(* IEC 61131-3 sources: SFWE411-511/ladder-diagrams/PLC/build/build, 2 files *)

(* ---- plc.st ---- *)
TYPE
  LOGLEVEL : (CRITICAL, WARNING, INFO, DEBUG) := INFO;
END_TYPE

FUNCTION_BLOCK LOGGER
  VAR_INPUT
    TRIG : BOOL;
    MSG : STRING;
    LEVEL : LOGLEVEL := INFO;
  END_VAR
  VAR
    TRIG0 : BOOL;
  END_VAR

  IF TRIG AND NOT TRIG0 THEN
  {{
   LogMessage(GetFbVar(LEVEL),(char*)GetFbVar(MSG, .body),GetFbVar(MSG, .len));
  }}
  END_IF;
  TRIG0:=TRIG;
END_FUNCTION_BLOCK

PROGRAM program0
  VAR
    EntranceGateSensor : BOOL;
    EntranceGateSensor0 : BOOL;
    ticketValidationEnter : BOOL;
    ticketValidationExit : BOOL;
    PhysicalCardEnter : BOOL;
    PhysicalCardExit : BOOL;
    PermitCardEnter : BOOL;
    PermitCardExit : BOOL;
    openSpotSensor : BOOL;
    countSensor : BOOL;
    overstayNotification : BOOL;
    OpenEntryGate : BOOL;
    OverstaySignage : BOOL;
    AvailableSpotSignage : BOOL;
    LicensePlateCapture : BOOL;
    LicensePlateVerification : BOOL;
    EntrancePassThrough : BOOL;
    AlarmButton : BOOL;
    TempSensor : BOOL;
    parkingLED : BOOL;
    AlarmActivate : BOOL;
    HealthDisplay : BOOL;
    CloseEntryGate : BOOL;
    LightSensor : INT := 100;
    SetLight : BOOL;
    RainSensor : BOOL;
    SnowSensor : BOOL;
    ClearWeather : BOOL;
    LightControl : BOOL;
    RainSignage : BOOL;
    SnowSignage : BOOL;
    ClearSignage : BOOL;
  END_VAR
  VAR
    ParkingTimer : INT;
    ParkingLimit : INT := 60;
  END_VAR
  VAR
    ParkingDurationStatus : BOOL;
    OverstayDetector : BOOL;
    TicketValidationSensor : BOOL;
    PaymentMachineDisplay : BOOL;
    EVSensorStatus : BOOL;
    EVChargerActivation : BOOL;
    ExitSensor : BOOL;
    ExitPassThroughSensor : BOOL;
    LicensePlateCaptureSystem : WORD;
    ExitGateOpens : BOOL;
    ExitGateCloses : BOOL;
  END_VAR
  VAR
    LightSensorCondition : INT := 10;
  END_VAR
  VAR
    HMIEntryDisplayTrigger : BOOL;
    OverstayPenaltyIndicator : BOOL;
    ParkingSpotDisplay : BOOL;
    AlarmStatusIndicator : BOOL;
    TemperatureDisplay : BOOL;
    LightningStatusDisplay : BOOL;
    WeatherConditionDisplay : BOOL;
    ParkingDurationOverstay : WORD;
    ExitEventDisplay : BOOL;
    PaymentProcessDisplay : BOOL;
    SystemHealthCheckDisplay : BOOL;
    ManualOverrideGate : BOOL;
    ManualOverrideAlarm : BOOL;
    ManualOverrideLight : BOOL;
    EventLogDisplay : BOOL;
    StatusSyncTrigger : BOOL;
    MaintenanceModeDisplay : BOOL;
  END_VAR
  VAR
    _TMP_LE61_OUT : BOOL;
    _TMP_GT41_OUT : BOOL;
  END_VAR

  OpenEntryGate := (PermitCardEnter OR PhysicalCardEnter OR ticketValidationEnter) AND EntranceGateSensor;
  CloseEntryGate := EntrancePassThrough;
  OverstaySignage := overstayNotification AND ticketValidationEnter;
  LicensePlateCapture := ticketValidationEnter AND EntranceGateSensor AND PhysicalCardEnter AND EntranceGateSensor AND PermitCardEnter AND EntranceGateSensor;
  AvailableSpotSignage := openSpotSensor;
  parkingLED := countSensor AND AvailableSpotSignage;
  AlarmActivate := AlarmButton;
  AlarmActivate := LicensePlateVerification;
  HealthDisplay := TempSensor;
  _TMP_LE61_OUT := LE(LightSensor, LightSensorCondition);
  LightControl := _TMP_LE61_OUT;
  RainSignage := RainSensor;
  SnowSignage := SnowSensor;
  ClearSignage := ClearWeather;
  _TMP_GT41_OUT := GT(ParkingTimer, ParkingLimit);
  ParkingDurationStatus := _TMP_GT41_OUT;
  overstayNotification := ParkingDurationStatus;
  EVChargerActivation := EVSensorStatus;
  LicensePlateCapture := ExitSensor;
  ExitGateOpens := (PermitCardExit OR PhysicalCardExit) AND ExitSensor;
  ExitGateCloses := ExitPassThroughSensor;
  TicketValidationSensor := ticketValidationExit;
  PaymentMachineDisplay := ticketValidationExit;
  ExitGateOpens := PaymentMachineDisplay;
  HMIEntryDisplayTrigger := LicensePlateCapture;
  OverstayPenaltyIndicator := overstayNotification AND ticketValidationEnter;
  AlarmStatusIndicator := AlarmButton;
  ParkingSpotDisplay := openSpotSensor;
  AlarmStatusIndicator := LicensePlateVerification;
  TemperatureDisplay := TempSensor;
  LightningStatusDisplay := _TMP_LE61_OUT;
  WeatherConditionDisplay := RainSensor;
  WeatherConditionDisplay := SnowSensor;
  WeatherConditionDisplay := ClearWeather;
  ParkingSpotDisplay := _TMP_GT41_OUT;
  OverstayPenaltyIndicator := ParkingDurationStatus;
  ExitEventDisplay := ExitSensor;
  ExitEventDisplay := PhysicalCardExit AND ExitSensor AND PermitCardExit AND ExitSensor;
  PaymentProcessDisplay := ticketValidationExit;
  PaymentProcessDisplay := ticketValidationExit;
  PaymentProcessDisplay := PaymentMachineDisplay;
  SystemHealthCheckDisplay := HealthDisplay;
  ManualOverrideAlarm := AlarmStatusIndicator;
  ManualOverrideGate := OpenEntryGate;
  EventLogDisplay := overstayNotification;
  StatusSyncTrigger := parkingLED;
  ManualOverrideLight := LightControl;
  ManualOverrideGate := ExitGateOpens;
END_PROGRAM

CONFIGURATION Config0

  RESOURCE Res0 ON PLC
    TASK task0(INTERVAL := T#20ms,PRIORITY := 0);
    PROGRAM instance0 WITH task0 : program0;
  END_RESOURCE
END_CONFIGURATION

(* ---- generated_plc.st ---- *)
PROGRAM program0
  VAR
    EntranceGateSensor AT %IX0.0 : BOOL;
    EntranceGateSensor0 AT %IX0.1 : BOOL;
    ticketValidationEnter AT %IX0.2 : BOOL;
    ticketValidationExit AT %IX2.4 : BOOL;
    PhysicalCardEnter AT %IX0.3 : BOOL;
    PhysicalCardExit AT %IX2.5 : BOOL;
    PermitCardEnter AT %IX0.7 : BOOL;
    PermitCardExit AT %IX2.6 : BOOL;
    openSpotSensor AT %IX1.1 : BOOL;
    countSensor AT %IX0.6 : BOOL;
    overstayNotification AT %IX0.5 : BOOL;
    OpenEntryGate AT %QX0.0 : BOOL;
    OverstaySignage AT %QX0.5 : BOOL;
    AvailableSpotSignage AT %QX0.8 : BOOL;
    LicensePlateCapture AT %IX1.0 : BOOL;
    LicensePlateVerification AT %IX5.1 : BOOL;
    EntrancePassThrough AT %IX0.8 : BOOL;
    AlarmButton AT %IX5.0 : BOOL;
    TempSensor AT %IX6.0 : BOOL;
    parkingLED AT %QX0.7 : BOOL;
    AlarmActivate AT %QX5.0 : BOOL;
    HealthDisplay AT %QX6.0 : BOOL;
    CloseEntryGate AT %QX0.6 : BOOL;
    LightSensor AT %IW2.0 : INT := 100;
    SetLight AT %IX2.4 : BOOL;
    RainSensor AT %IX2.1 : BOOL;
    SnowSensor AT %IX2.2 : BOOL;
    ClearWeather AT %IX2.3 : BOOL;
    LightControl AT %QX2.0 : BOOL;
    RainSignage AT %QX2.1 : BOOL;
    SnowSignage AT %QX2.2 : BOOL;
    ClearSignage AT %QX2.3 : BOOL;
  END_VAR
  VAR
    ParkingTimer : INT;
    ParkingLimit : INT := 60;
  END_VAR
  VAR
    ParkingDurationStatus AT %QX3.0 : BOOL;
    OverstayDetector AT %IX3.1 : BOOL;
    TicketValidationSensor AT %QX3.2 : BOOL;
    PaymentMachineDisplay AT %QX3.3 : BOOL;
    EVSensorStatus AT %IX4.0 : BOOL;
    EVChargerActivation AT %QX4.0 : BOOL;
    ExitSensor AT %IX0.4 : BOOL;
    ExitPassThroughSensor AT %IX0.8 : BOOL;
    LicensePlateCaptureSystem AT %QW0.1 : WORD;
    ExitGateOpens AT %QX0.4 : BOOL;
    ExitGateCloses AT %QX0.9 : BOOL;
  END_VAR
  VAR
    LightSensorCondition : INT := 10;
  END_VAR
  VAR
    HMIEntryDisplayTrigger AT %QX7.0 : BOOL;
    OverstayPenaltyIndicator AT %QX7.1 : BOOL;
    ParkingSpotDisplay AT %QW7.2 : BOOL;
    AlarmStatusIndicator AT %QX7.3 : BOOL;
    TemperatureDisplay AT %QW7.4 : BOOL;
    LightningStatusDisplay AT %QX7.5 : BOOL;
    WeatherConditionDisplay AT %QW7.6 : BOOL;
    ParkingDurationOverstay AT %QW7.7 : WORD;
    ExitEventDisplay AT %QX8.0 : BOOL;
    PaymentProcessDisplay AT %QW8.1 : BOOL;
    SystemHealthCheckDisplay AT %QX8.2 : BOOL;
    ManualOverrideGate AT %QX8.3 : BOOL;
    ManualOverrideAlarm AT %QX8.4 : BOOL;
    ManualOverrideLight AT %QX8.5 : BOOL;
    EventLogDisplay AT %QW8.6 : BOOL;
    StatusSyncTrigger AT %QX8.7 : BOOL;
    MaintenanceModeDisplay AT %QX9.0 : BOOL;
  END_VAR
  VAR
    _TMP_LE61_OUT : BOOL;
    _TMP_GT41_OUT : BOOL;
  END_VAR

  OpenEntryGate := (PermitCardEnter OR PhysicalCardEnter OR ticketValidationEnter) AND EntranceGateSensor;
  CloseEntryGate := EntrancePassThrough;
  OverstaySignage := overstayNotification AND ticketValidationEnter;
  LicensePlateCapture := ticketValidationEnter AND EntranceGateSensor AND PhysicalCardEnter AND EntranceGateSensor AND PermitCardEnter AND EntranceGateSensor;
  AvailableSpotSignage := openSpotSensor;
  parkingLED := countSensor AND AvailableSpotSignage;
  AlarmActivate := AlarmButton;
  AlarmActivate := LicensePlateVerification;
  HealthDisplay := TempSensor;
  _TMP_LE61_OUT := LE(LightSensor, LightSensorCondition);
  LightControl := _TMP_LE61_OUT;
  RainSignage := RainSensor;
  SnowSignage := SnowSensor;
  ClearSignage := ClearWeather;
  _TMP_GT41_OUT := GT(ParkingTimer, ParkingLimit);
  ParkingDurationStatus := _TMP_GT41_OUT;
  overstayNotification := ParkingDurationStatus;
  EVChargerActivation := EVSensorStatus;
  LicensePlateCapture := ExitSensor;
  ExitGateOpens := (PermitCardExit OR PhysicalCardExit) AND ExitSensor;
  ExitGateCloses := ExitPassThroughSensor;
  TicketValidationSensor := ticketValidationExit;
  PaymentMachineDisplay := ticketValidationExit;
  ExitGateOpens := PaymentMachineDisplay;
  HMIEntryDisplayTrigger := LicensePlateCapture;
  OverstayPenaltyIndicator := overstayNotification AND ticketValidationEnter;
  AlarmStatusIndicator := AlarmButton;
  ParkingSpotDisplay := openSpotSensor;
  AlarmStatusIndicator := LicensePlateVerification;
  TemperatureDisplay := TempSensor;
  LightningStatusDisplay := _TMP_LE61_OUT;
  WeatherConditionDisplay := RainSensor;
  WeatherConditionDisplay := SnowSensor;
  WeatherConditionDisplay := ClearWeather;
  ParkingSpotDisplay := _TMP_GT41_OUT;
  OverstayPenaltyIndicator := ParkingDurationStatus;
  ExitEventDisplay := ExitSensor;
  ExitEventDisplay := PhysicalCardExit AND ExitSensor AND PermitCardExit AND ExitSensor;
  PaymentProcessDisplay := ticketValidationExit;
  PaymentProcessDisplay := ticketValidationExit;
  PaymentProcessDisplay := PaymentMachineDisplay;
  SystemHealthCheckDisplay := HealthDisplay;
  ManualOverrideAlarm := AlarmStatusIndicator;
  ManualOverrideGate := OpenEntryGate;
  EventLogDisplay := overstayNotification;
  StatusSyncTrigger := parkingLED;
  ManualOverrideLight := LightControl;
  ManualOverrideGate := ExitGateOpens;
END_PROGRAM

CONFIGURATION Config0

  RESOURCE Res0 ON PLC
    TASK task0(INTERVAL := T#20ms,PRIORITY := 0);
    PROGRAM instance0 WITH task0 : program0;
  END_RESOURCE
END_CONFIGURATION
